TYPE ST_Camera_CycleData :
STRUCT
	/////////////////////////////////////////////////////////////////////////////////////SETTINGS/////////////////////////////////////////////////////////////////////////////////////			
(**************************************************************************CURRENT SETTINGS DURING CYCLE. VELOCITY FOR EXAMPLE****************************************************)	
	
	anDistanceCalibrationBlock				: ARRAY [0..2] OF DINT;	
	anExpectedDistances						: ARRAY [0..2] OF DINT;	
	anHeightSetByCalibration				: ARRAY [0..3] OF DINT;	
	anTolerances							: ARRAY [0..2] OF DINT;	
	
	
/////////////////////////////////////////////////////////////////////////////////////GENERAL DATA/////////////////////////////////////////////////////////////////////////////////////			
(**************************************************************************RESULT DATA OF THE CYCLE. DISTANCE FOR EXAMPLE************************************************************)	
	
	anDistancesResult						: ARRAY [0..2] OF DINT;

////////////////////////////////////////////////////////////////////////////////////RESULTS////////////////////////////////////////////////////////////////////////////////////////
(**************************************************************************DETERMINE IF THE PART FAIL OR PASS*********************************************************************)

	bPass				: BOOL;
	bFail				: BOOL;		

END_STRUCT
END_TYPE

(* stored: Version 1.1.0.1, ProductVersion 3.1.4024.13
   DUT ST_Camera_CycleData: Id {5b94fbf5-07bd-473e-8e05-f4b5f00f766b} *)
